{attribute 'GeneratedUsingTerminal: EL6784-0000-0016'}
{attribute addProperty BoxType "EL6784-0000-0016"}
{attribute addProperty Id "EtcSlaveTerminalBaseStatusAT %I*Status_07D3AAF62InputsEMPTY_STRUCTURE0ControlAT %Q*Control_DAFD38E02OutputsEMPTY_STRUCTURE0WcStateAT %I*WcState_9091E0EB2InfoDataAT %I*InfoData_32EB74EA10"}
{attribute addProperty CRC "3129702536"}
{attribute addProperty Size "16"}
TYPE EL6784_BA8B7888 EXTENDS EtcSlaveTerminalBase :
STRUCT
	{attribute addProperty Name "Status"}
	Status : Status_07D3AAF6;
	{attribute addProperty Name "Inputs"}
	Inputs : EMPTY_STRUCTURE;
	{attribute addProperty Name "Control"}
	Control : Control_DAFD38E0;
	{attribute addProperty Name "Outputs"}
	Outputs : EMPTY_STRUCTURE;
	{attribute addProperty Name "WcState"}
	WcState : WcState_9091E0EB;
	{attribute addProperty Name "InfoData"}
	InfoData : InfoData_32EB74EA;
END_STRUCT
END_TYPE

(* stored: Version 1.2.0.0, ProductVersion 3.1.4024.9
   DUT EL6784_BA8B7888: Id {ccbb5d21-d1ca-445f-95bb-42098fdd2ce9} *)
